Staubli VAL3: start.pgx

public program start()
begin
  nBuffer = 0
  nNum = 0
  nFailCounter = 0
  bDetectInput = false
  sInput = ""
  //call enablePowerTest()
  call detectInput()
end
